SUBAPPLICATION Uebung_247_AX (* Wie Uebung_245_AX (Korrekturfaktor via AR_MUL_2/initval_AR), zusaetzlich echter logiBUS_QDA_PWM-Ausgang Q1 zum Nachmessen *)
  (* Standard: 61499-2; Description: Copyright (c) 2026 Meisterschulen am Ostbahnhof This program and the accompanying materials are made available under the terms of the Eclipse Public License 2.0 which is available at https://www.eclipse.org/legal/epl-2.0/ SPDX-License-Identifier: EPL-2.0 *)
  (* Version 1.0, 2026-09-07, Franz Höpfinger, Meisterschulen am Ostbahnhof, initial API and implementation and/or initial documentation *)
  PACKAGE Uebungen;
  IMPORT Uebungen::const::UT::DefaultPool_Numeric::InputNumber_I3_N;
  IMPORT Uebungen::const::UT::DefaultPool_Numeric::OutputNumber_N3_N;
  IMPORT logiBUS::io::DQ::logiBUS_DO::Output_Q1;
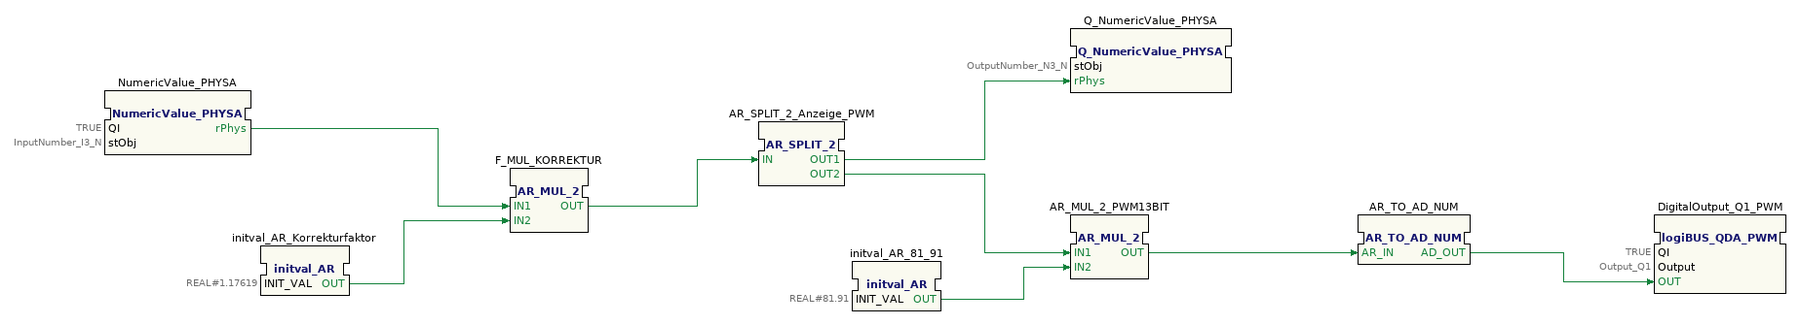
  (* 0-100% Tastgrad = 0-8191 (13-Bit LEDC, siehe RampLimitFS_TO_logiBUS_QDA_PWM_OPC.SUB in MyLib_AX-1.0.0): Faktor 81,91 = 8191/100. Korrigierter Wert (bis 117,619% bei I3>85%) wird NICHT geklemmt - zum Nachmessen absichtlich so belassen, siehe Beschreibung. Mit Multimeter/Oszilloskop an Q1 gegen GND: Mittelwert = Tastgrad% x Versorgungsspannung. *)
  FBS
    NumericValue_PHYSA : isobus::UT::io::NumericValue::NumericValue_PHYSA(QI := TRUE, stObj := InputNumber_I3_N);
    F_MUL_KORREKTUR : adapter::iec61131::arithmetic::AR_MUL_2;
    initval_AR_Korrekturfaktor : adapter::types::unidirectional::AR::initval::initval_AR(INIT_VAL := REAL#1.17619);
    AR_SPLIT_2_Anzeige_PWM : adapter::events::unidirectional::AR_SPLIT_2;
    Q_NumericValue_PHYSA : isobus::UT::Q::Q_NumericValue_PHYSA(stObj := OutputNumber_N3_N);
    AR_MUL_2_PWM13BIT : adapter::iec61131::arithmetic::AR_MUL_2;
    initval_AR_81_91 : adapter::types::unidirectional::AR::initval::initval_AR(INIT_VAL := REAL#81.91);
    DigitalOutput_Q1_PWM : logiBUS::io::DQ::logiBUS_QDA_PWM(QI := TRUE, Output := Output_Q1);
    AR_TO_AD_NUM : adapter::conversion::unidirectional::AR_TO_AD_NUM;
  END_FBS
  ADAPTER_CONNECTIONS
    NumericValue_PHYSA.rPhys TO F_MUL_KORREKTUR.IN1;
    initval_AR_Korrekturfaktor.OUT TO F_MUL_KORREKTUR.IN2;
    F_MUL_KORREKTUR.OUT TO AR_SPLIT_2_Anzeige_PWM.IN;
    AR_SPLIT_2_Anzeige_PWM.OUT1 TO Q_NumericValue_PHYSA.rPhys;
    AR_SPLIT_2_Anzeige_PWM.OUT2 TO AR_MUL_2_PWM13BIT.IN1;
    initval_AR_81_91.OUT TO AR_MUL_2_PWM13BIT.IN2;
    AR_MUL_2_PWM13BIT.OUT TO AR_TO_AD_NUM.AR_IN;
    AR_TO_AD_NUM.AD_OUT TO DigitalOutput_Q1_PWM.OUT;
  END_CONNECTIONS
END_SUBAPPLICATION
